{attribute addProperty BoxType "EPP3204-0002-0017"}
{attribute addProperty Id "RTD_RTDInputs_ChannelAT %I*ARRAY[0..6] OF RTD_RTDInputs_Channel_F16A160D128160WcStateAT %I*WcState_98A4DF7520.250InfoDataAT %I*InfoData_BC63D37F80100"}
{attribute addProperty CRC "216835468"}
{attribute addProperty SizeInBites "210"}
{attribute addProperty SizeInBytes "26.25"}
TYPE EPP3204_C91659E2 :
STRUCT
	{attribute addProperty Name "RTD_RTDInputs_Channel"}
	RTD_RTDInputs_Channel : ARRAY[0..6] OF RTD_RTDInputs_Channel_F16A160D;
	{attribute addProperty Name "WcState"}
	WcState : WcState_98A4DF75;
	{attribute addProperty Name "InfoData"}
	InfoData : InfoData_BC63D37F;
END_STRUCT
END_TYPE

(* stored: Version 1.2.0.0, ProductVersion 3.1.4024.9
   DUT EPP3204_C91659E2: Id {09e46609-8f0a-47b6-9e92-729f2bf0a902} *)
